// TwinCAT 3 PLC project kfe_rix_motion
// Title: plc-kfe-rix-motion
// Company: SLAC
// ProjectVersion: 0.0.0
// ProgramVersion: 3.1.4022.7
// CompilerDefines: K
// libraries:
//   LCLS General, * (SLAC)
//   lcls-twincat-common-components, * (SLAC)
//   lcls-twincat-motion, * (SLAC)
//   lcls-twincat-physics, * (SLAC)
//   PMPS, * (SLAC - LCLS)
//   Tc2_Standard, * (Beckhoff Automation GmbH)
//   Tc2_System, * (Beckhoff Automation GmbH)
//   Tc3_Module, * (Beckhoff Automation GmbH)
// project tree:
//   DUTs/ DUT_SATT_Filter.TcDUT (not stored), ENUM_SXR_SATT_Position.TcDUT (not stored)
//   GVLs/ GVL.TcGVL (not stored), Main.TcGVL (not stored)
//   / PlcTask.TcTTO (not stored)
//   POUs/AT1K2/ FB_AT1K2.TcPOU (not stored)
//   POUs/AT2K2/ FB_AttenuatorElementDensity.TcPOU (not stored), FB_SXR_SATT_PositionState.TcPOU (not stored), FB_SXR_SATT_Stage.TcPOU (not stored)
//   POUs/ PRG_1_PlcTask.TcPOU (not stored), PRG_2_PMPS_PRE.TcPOU (not stored), PRG_3_PMPS_POST.TcPOU (not stored), PRG_4_LOG.TcPOU (not stored), PRG_AT1K2_SOLID.TcPOU (not stored), PRG_AT2K2_SOLID.TcPOU (not stored), PRG_IM6K2_PPM.TcPOU, PRG_LI3K2_K2B.TcPOU, PRG_PF1K2_WFS.TcPOU, PRG_LI2K2_K2A.TcPOU, PRG_IM1K1_PPM.TcPOU, PRG_AL1K2_L2SI.TcPOU, PRG_IM2K2_PPM.TcPOU, PRG_IM2K1_PPM.TcPOU, PRG_IM1K2_PPM.TcPOU, PRG_IM3K2_PPM.TcPOU, PRG_IM4K2_PPM.TcPOU, PRG_IM5K2_PPM.TcPOU, PRG_PF2K2_WFS.TcPOU, PRG_TM1K2_ATM.TcPOU, PRG_TM2K2_ATM.TcPOU (not stored), PRG_ST3K2_TERM.TcPOU (not stored)
//   POUs/TM2K2/ ENUM_TM2K2_States.TcDUT (not stored), FB_TM2K2.TcPOU (not stored), FB_TM2K2_States.TcPOU (not stored)

// ---- POUs/PRG_IM6K2_PPM.TcPOU
PROGRAM PRG_IM6K2_PPM
VAR
    {attribute 'pytmc' := '
        pv: IM6K2:PPM
        io: io
    '}
    {attribute 'TcLinkTo' := '.fbGige.iIlluminatorINT := TIIB[IM6K2-EL4004-E7]^AO Outputs Channel 1^Analog output;
                              .fbGige.bGigePower := TIIB[IM6K2-EL2004-E3]^Channel 2^Output;
                              .fbPowerMeter.iVoltageINT := TIIB[IM6K2-EL3062-E6]^AI Standard Channel 1^Value;
                              .fbPowerMeter.fbThermoCouple.bError := TIIB[IM6K2-EL3314-E4]^TC Inputs Channel 1^Status^Error;
                              .fbPowerMeter.fbThermoCouple.bUnderrange := TIIB[IM6K2-EL3314-E4]^TC Inputs Channel 1^Status^Underrange;
                              .fbPowerMeter.fbThermoCouple.bOverrange := TIIB[IM6K2-EL3314-E4]^TC Inputs Channel 1^Status^Overrange;
                              .fbPowerMeter.fbThermoCouple.iRaw := TIIB[IM6K2-EL3314-E4]^TC Inputs Channel 1^Value;
                              .fbYagThermoCouple.bError := TIIB[IM6K2-EL3314-E4]^TC Inputs Channel 2^Status^Error;
                              .fbYagThermoCouple.bUnderrange := TIIB[IM6K2-EL3314-E4]^TC Inputs Channel 2^Status^Underrange;
                              .fbYagThermoCouple.bOverrange := TIIB[IM6K2-EL3314-E4]^TC Inputs Channel 2^Status^Overrange;
                              .fbYagThermoCouple.iRaw 6K2-EL3314-E4]^TC Inputs Channel 2^Value;
                              .fbFlowMeter.iRaw := TIIB[IM1K2-EL3052-E5]^AI Standard Channel 1^Value'}
    fbIM6K2: FB_PPM;
END_VAR


fbIM6K2.stOut.fPosition := -8.61;
fbIM6K2.stOut.bUseRawCounts := FALSE;
fbIM6K2.stOut.bValid := TRUE;
fbIM6K2.stOut.stPMPS.sPmpsState := 'IM6K2:PPM-OUT';

fbIM6K2.stPower.fPosition := -47.71;
fbIM6K2.stPower.bUseRawCounts := FALSE;
fbIM6K2.stPower.bValid := TRUE;
fbIM6K2.stPower.stPMPS.sPmpsState := 'IM6K2:PPM-POWERMETER';

fbIM6K2.stYag1.fPosition := -71.71;
fbIM6K2.stYag1.bUseRawCounts := FALSE;
fbIM6K2.stYag1.bValid := TRUE;
fbIM6K2.stYag1.stPMPS.sPmpsState := 'IM6K2:PPM-YAG1';

fbIM6K2.stYag2.fPosition := -97.72;
fbIM6K2.stYag2.bUseRawCounts := FALSE;
fbIM6K2.stYag2.bValid := TRUE;
fbIM6K2.stYag2.stPMPS.sPmpsState := 'IM6K2:PPM-YAG2';

fbIM6K2(
    fbArbiter := GVL.fbArbiter2,
    fbFFHWO := GVL.fbFastFaultOutput2,
    stYStage := Main.M24,
    sDeviceName := 'IM6K2:PPM',
    sTransitionKey := 'IM6K2:PPM-TRANSITION',
    bEnableMotion := TRUE,
    bEnableBeamParams := TRUE,
    bEnablePositionLimits := TRUE,
    fFlowOffset := 0.0,
);

END_PROGRAM

// ---- POUs/PRG_LI3K2_K2B.TcPOU
PROGRAM PRG_LI3K2_K2B
VAR
    {attribute 'pytmc' := '
        pv: LI3K2:K2B
        io: io
    '}
    fbLI3K2: FB_LIC;

    //stSiBP: ST_BeamParams := PMPS_GVL.cstFullBeam;
    //stFoilBP: ST_BeamParams := PMPS_GVL.cstFullBeam;
END_VAR

(*
   Avoid damage peak between 3.2 keV and 1.6 keV
*)
//stSiBp.neVRange := F_eVExcludeRange(1600, 3200);
// Drop transmission to 20%
//stSiBP.nTran := 0.2;

// Drop transmission to 10%
//stFoilBP.nTran := 0.1;

fbLI3K2.stOut.fPosition := 0.118;
fbLI3K2.stOut.bUseRawCounts := FALSE;
fbLI3K2.stOut.bValid := TRUE;
fbLI3K2.stOut.stPMPS.sPmpsState := 'LI3K2:K2B-OUT';

fbLI3K2.stMirror1.fPosition := -36.38;
fbLI3K2.stMirror1.bUseRawCounts := FALSE;
fbLI3K2.stMirror1.bValid := TRUE;
fbLI3K2.stMirror1.stPMPS.sPmpsState := 'LI3K2:K2B-MIRROR1';

fbLI3K2.stMirror2.fPosition := -70.38;
fbLI3K2.stMirror2.bUseRawCounts := FALSE;
fbLI3K2.stMirror2.bValid := TRUE;
fbLI3K2.stMirror2.stPMPS.sPmpsState := 'LI3K2:K2B-MIRROR2';

fbLI3K2.stTarget1.fPosition := -102.38;
fbLI3K2.stTarget1.bUseRawCounts := FALSE;
fbLI3K2.stTarget1.bValid := TRUE;
fbLI3K2.stTarget1.stPMPS.sPmpsState := 'LI3K2:K2B-TARGET1';

fbLI3K2(
    fbArbiter := GVL.fbArbiter2,
    fbFFHWO := GVL.fbFastFaultOutput2,
    stYStage := Main.M21,
    sDeviceName := 'LI3K2:K2B',
    sTransitionKey := 'LI3K2:K2B-TRANSITION',
    bEnableMotion := TRUE,
    bEnableBeamParams := TRUE,
    bEnablePositionLimits := TRUE,
);

END_PROGRAM

// ---- POUs/PRG_PF1K2_WFS.TcPOU
PROGRAM PRG_PF1K2_WFS
VAR
    {attribute 'pytmc' := '
        pv: PF1K2:WFS
        io: io
    '}
    {attribute 'TcLinkTo' := '.fbThermoCouple1.bError 		:= TIIB[PF1K2-EL3314-E5]^TC Inputs Channel 1^Status^Error;
                              .fbThermoCouple1.bUnderrange	:= TIIB[PF1K2-EL3314-E5]^TC Inputs Channel 1^Status^Underrange;
                              .fbThermoCouple1.bOverrange 	:= TIIB[PF1K2-EL3314-E5]^TC Inputs Channel 1^Status^Overrange;
                              .fbThermoCouple1.iRaw 		:= TIIB[PF1K2-EL3314-E5]^TC Inputs Channel 1^Value;
                              .fbThermoCouple2.bError 		:= TIIB[PF1K2-EL3314-E5]^TC Inputs Channel 2^Status^Error;
                              .fbThermoCouple2.bUnderrange 	:= TIIB[PF1K2-EL3314-E5]^TC Inputs Channel 2^Status^Underrange;
                              .fbThermoCouple2.bOverrange 	:= TIIB[PF1K2-EL3314-E5]^TC Inputs Channel 2^Status^Overrange;
                              .fbThermoCouple2.iRaw 		:= TIIB[PF1K2-EL3314-E5]^TC Inputs Channel 2^Value'}
    fbPF1K2: FB_WFS;

    //stSiBP: ST_BeamParams := PMPS_GVL.cstFullBeam;
END_VAR

(*
   Avoid damage peak between 3.2 keV and 1.6 keV
*)
//stSiBp.neVRange := F_eVExcludeRange(1600, 3200);
// Drop transmission to 20%
//stSiBP.nTran := 0.2;

fbPF1K2.stOut.fPosition := -13.00;
fbPF1K2.stOut.bUseRawCounts := FALSE;
fbPF1K2.stOut.bValid := TRUE;
fbPF1K2.stOut.stPMPS.sPmpsState := 'PF1K2:WFS-OUT';

fbPF1K2.stTarget1.fPosition := -97.13;
fbPF1K2.stTarget1.bUseRawCounts := FALSE;
fbPF1K2.stTarget1.bValid := TRUE;
fbPF1K2.stTarget1.stPMPS.sPmpsState := 'PF1K2:WFS-TARGET1';

fbPF1K2.stTarget2.fPosition := -82.755;
fbPF1K2.stTarget2.bUseRawCounts := FALSE;
fbPF1K2.stTarget2.bValid := TRUE;
fbPF1K2.stTarget2.stPMPS.sPmpsState := 'PF1K2:WFS-TARGET2';

fbPF1K2.stTarget3.fPosition := -68.38;
fbPF1K2.stTarget3.bUseRawCounts := FALSE;
fbPF1K2.stTarget3.bValid := TRUE;
fbPF1K2.stTarget3.stPMPS.sPmpsState := 'PF1K2:WFS-TARGET3';

fbPF1K2.stTarget4.fPosition := -54.004;
fbPF1K2.stTarget4.bUseRawCounts := FALSE;
fbPF1K2.stTarget4.bValid := TRUE;
fbPF1K2.stTarget4.stPMPS.sPmpsState := 'PF1K2:WFS-TARGET4';

fbPF1K2.stTarget5.fPosition := -39.629;
fbPF1K2.stTarget5.bUseRawCounts := FALSE;
fbPF1K2.stTarget5.bValid := TRUE;
fbPF1K2.stTarget5.stPMPS.sPmpsState := 'PF1K2:WFS-TARGET5';

fbPF1K2(
    fbArbiter := GVL.fbArbiter2,
    fbFFHWO := GVL.fbFastFaultOutput2,
    stYStage := Main.M12,
    stZStage := Main.M13,
    sDeviceName := 'PF1K2:WFS',
    sTransitionKey := 'PF1K2:WFS-TRANSITION',
    bEnableMotion := TRUE,
    bEnableBeamParams := TRUE,
    bEnablePositionLimits := TRUE,
);

END_PROGRAM

// ---- POUs/PRG_LI2K2_K2A.TcPOU
PROGRAM PRG_LI2K2_K2A
VAR
    {attribute 'pytmc' := '
        pv: LI2K2:K2A
        io: io
    '}
    fbLI2K2: FB_LIC;

    //stSiBP: ST_BeamParams := PMPS_GVL.cstFullBeam;
    //stFoilBP: ST_BeamParams := PMPS_GVL.cstFullBeam;
END_VAR

(*
   Avoid damage peak between 3.2 keV and 1.6 keV
*)
//stSiBp.neVRange := F_eVExcludeRange(1600, 3200);
// Drop transmission to 20%
//stSiBP.nTran := 0.2;

// Drop transmission to 10%
////stFoilBP.nTran := 0.1;

fbLI2K2.stOut.fPosition := 1.2;
fbLI2K2.stOut.bUseRawCounts := FALSE;
fbLI2K2.stOut.bValid := TRUE;
fbLI2K2.stOut.stPMPS.sPmpsState := 'LI2K2:K2A-OUT';

fbLI2K2.stMirror1.fPosition := -35.3;
fbLI2K2.stMirror1.bUseRawCounts := FALSE;
fbLI2K2.stMirror1.bValid := TRUE;
fbLI2K2.stMirror1.stPMPS.sPmpsState := 'LI2K2:K2A-MIRROR1';

fbLI2K2.stMirror2.fPosition := -69.3;
fbLI2K2.stMirror2.bUseRawCounts := FALSE;
fbLI2K2.stMirror2.bValid := TRUE;
fbLI2K2.stMirror2.stPMPS.sPmpsState := 'LI2K2:K2A-MIRROR2';

fbLI2K2.stTarget1.fPosition := -101.3;
fbLI2K2.stTarget1.bUseRawCounts := FALSE;
fbLI2K2.stTarget1.bValid := TRUE;
fbLI2K2.stTarget1.stPMPS.sPmpsState := 'LI2K2:K2A-TARGET1';

fbLI2K2(
    fbArbiter := GVL.fbArbiter2,
    fbFFHWO := GVL.fbFastFaultOutput2,
    stYStage := Main.M11,
    sDeviceName := 'LI2K2:K2A',
    sTransitionKey := 'LI2K2:K2A-TRANSITION',
    bEnableMotion := TRUE,
    bEnableBeamParams := TRUE,
    bEnablePositionLimits := TRUE,
);

END_PROGRAM

// ---- POUs/PRG_IM1K1_PPM.TcPOU
PROGRAM PRG_IM1K1_PPM
VAR
    {attribute 'pytmc' := '
        pv: IM1K1:PPM
        io: io
    '}
    {attribute 'TcLinkTo' := '.fbGige.iIlluminatorINT := TIIB[IM1K1-EL4004]^AO Outputs Channel 1^Analog output;
                              .fbGige.bGigePower := TIIB[IM1K1-EL2004]^Channel 2^Output;
                              .fbPowerMeter.iVoltageINT := TIIB[IM1K1-EL3062]^AI Standard Channel 1^Value;
                              .fbPowerMeter.fbThermoCouple.bError := TIIB[IM1K1-EL3314]^TC Inputs Channel 1^Status^Error;
                              .fbPowerMeter.fbThermoCouple.bUnderrange := TIIB[IM1K1-EL3314]^TC Inputs Channel 1^Status^Underrange;
                              .fbPowerMeter.fbThermoCouple.bOverrange := TIIB[IM1K1-EL3314]^TC Inputs Channel 1^Status^Overrange;
                              .fbPowerMeter.fbThermoCouple.iRaw := TIIB[IM1K1-EL3314]^TC Inputs Channel 1^Value;
                              .fbYagThermoCouple.bError := TIIB[IM1K1-EL3314]^TC Inputs Channel 2^Status^Error;
                              .fbYagThermoCouple.bUnderrange := TIIB[IM1K1-EL3314]^TC Inputs Channel 2^Status^Underrange;
                              .fbYagThermoCouple.bOverrange := TIIB[IM1K1-EL3314]^TC Inputs Channel 2^Status^Overrange;
                              .fbYagThermoCouple.iRaw := TIIB[IM1K1-EL3314]^TC Inputs Channel 2^Value'}
    fbIM1K1: FB_PPM;
END_VAR

fbIM1K1.stOut.fPosition := -8.82;
fbIM1K1.stOut.bUseRawCounts := FALSE;
fbIM1K1.stOut.bValid := TRUE;
fbIM1K1.stOut.stPMPS.sPmpsState := 'IM1K1:PPM-OUT';

fbIM1K1.stPower.fPosition := -47.92;
fbIM1K1.stPower.bUseRawCounts := FALSE;
fbIM1K1.stPower.bValid := TRUE;
fbIM1K1.stPower.stPMPS.sPmpsState := 'IM1K1:PPM-POWERMETER';

fbIM1K1.stYag1.fPosition := -71.92;
fbIM1K1.stYag1.bUseRawCounts := FALSE;
fbIM1K1.stYag1.bValid := TRUE;
fbIM1K1.stYag1.stPMPS.sPmpsState := 'IM1K1:PPM-YAG1';

fbIM1K1.stYag2.fPosition := -97.93;
fbIM1K1.stYag2.bUseRawCounts := FALSE;
fbIM1K1.stYag2.bValid := TRUE;
fbIM1K1.stYag2.stPMPS.sPmpsState := 'IM1K1:PPM-YAG2';

fbIM1K1(
    fbArbiter := GVL.fbArbiter1,
    fbFFHWO := GVL.fbFastFaultOutput1,
    stYStage := Main.M1,
    sDeviceName := 'IM1K1:PPM',
    sTransitionKey := 'IM1K1:PPM-TRANSITION',
    bEnableMotion := TRUE,
    bEnableBeamParams := TRUE,
    bEnablePositionLimits := FALSE,
    fFlowOffset := 0.0,
);

END_PROGRAM

// ---- POUs/PRG_AL1K2_L2SI.TcPOU
PROGRAM PRG_AL1K2_L2SI
VAR
    {attribute 'pytmc' := '
        pv: AL1K2:L2SI
        io: io
    '}
    {attribute 'TcLinkTo' := '.fbLaser.iLaserINT := TIIB[AL1K2-EL4004-E4]^AO Outputs Channel 1^Analog output;
                              .fbLaser.iShutdownINT := TIIB[AL1K2-EL4004-E4]^AO Outputs Channel 2^Analog output'}
    fbAL1K2: FB_REF;
END_VAR


fbAL1K2.stOut.fPosition := -33.5; // Upper limit
fbAL1K2.stOut.bUseRawCounts := FALSE;
fbAL1K2.stOut.bValid := TRUE;
fbAL1K2.stOut.stPMPS.sPmpsState := 'AL1K2:L2SI-OUT';

fbAL1K2.stIn.fPosition := -75; // Current position at time of edit
fbAL1K2.stIn.bUseRawCounts := FALSE;
fbAL1K2.stIn.bValid := TRUE;
fbAL1K2.stIn.stPMPS.sPmpsState := 'AL1K2:L2SI-IN';

fbAL1K2(
    stYStage := Main.M5,
    fbArbiter := GVL.fbArbiter2,
    fbFFHWO := GVL.fbFastFaultOutput2,
    sDeviceName := 'AL1K2:L2SI',
    sTransitionKey := 'AL1K2:L2SI-TRANSITION',
    bEnableMotion := TRUE,
    bEnableBeamParams := TRUE,
    bEnablePositionLimits := TRUE
);

END_PROGRAM

// ---- POUs/PRG_IM2K2_PPM.TcPOU
PROGRAM PRG_IM2K2_PPM
VAR
    {attribute 'pytmc' := '
        pv: IM2K2:PPM
        io: io
    '}
    {attribute 'TcLinkTo' := '.fbGige.iIlluminatorINT := TIIB[IM2K2-EL4004-E7]^AO Outputs Channel 1^Analog output;
                              .fbGige.bGigePower := TIIB[IM2K2-EL2004-E3]^Channel 2^Output;
                              .fbPowerMeter.iVoltageINT := TIIB[IM2K2-EL3062-E6]^AI Standard Channel 1^Value;
                              .fbPowerMeter.fbThermoCouple.bError := TIIB[IM2K2-EL3314-E4]^TC Inputs Channel 1^Status^Error;
                              .fbPowerMeter.fbThermoCouple.bUnderrange := TIIB[IM2K2-EL3314-E4]^TC Inputs Channel 1^Status^Underrange;
                              .fbPowerMeter.fbThermoCouple.bOverrange := TIIB[IM2K2-EL3314-E4]^TC Inputs Channel 1^Status^Overrange;
                              .fbPowerMeter.fbThermoCouple.iRaw := TIIB[IM2K2-EL3314-E4]^TC Inputs Channel 1^Value;
                              .fbYagThermoCouple.bError := TIIB[IM2K2-EL3314-E4]^TC Inputs Channel 2^Status^Error;
                              .fbYagThermoCouple.bUnderrange := TIIB[IM2K2-EL3314-E4]^TC Inputs Channel 2^Status^Underrange;
                              .fbYagThermoCouple.bOverrange := TIIB[IM2K2-EL3314-E4]^TC Inputs Channel 2^Status^Overrange;
                              .fbYagThermoCouple.iRaw := TIIB[IM2K2-EL3314-E4]^TC Inputs Channel 2^Value;
                              .fbFlowMeter.iRaw := TIIB[IM1K2-EL3052-E5]^AI Standard Channel 1^Value'}  //IM1/2/3/4K2 same flow meter
    fbIM2K2: FB_PPM;
END_VAR


fbIM2K2.stOut.fPosition := -8.49;
fbIM2K2.stOut.bUseRawCounts := FALSE;
fbIM2K2.stOut.bValid := TRUE;
fbIM2K2.stOut.stPMPS.sPmpsState := 'IM2K2:PPM-OUT';

fbIM2K2.stPower.fPosition := -47.59;
fbIM2K2.stPower.bUseRawCounts := FALSE;
fbIM2K2.stPower.bValid := TRUE;
fbIM2K2.stPower.stPMPS.sPmpsState := 'IM2K2:PPM-POWERMETER';

fbIM2K2.stYag1.fPosition := -71.59;
fbIM2K2.stYag1.bUseRawCounts := FALSE;
fbIM2K2.stYag1.bValid := TRUE;
fbIM2K2.stYag1.stPMPS.sPmpsState := 'IM2K2:PPM-YAG1';

fbIM2K2.stYag2.fPosition := -97.60;
fbIM2K2.stYag2.bUseRawCounts := FALSE;
fbIM2K2.stYag2.bValid := TRUE;
fbIM2K2.stYag2.stPMPS.sPmpsState := 'IM2K2:PPM-YAG2';

fbIM2K2(
    fbArbiter := GVL.fbArbiter2,
    fbFFHWO := GVL.fbFastFaultOutput2,
    stYStage := Main.M6,
    sDeviceName := 'IM2K2:PPM',
    sTransitionKey := 'IM2K2:PPM-TRANSITION',
    bEnableMotion := TRUE,
    bEnableBeamParams := TRUE,
    bEnablePositionLimits := TRUE,
);

END_PROGRAM

// ---- POUs/PRG_IM2K1_PPM.TcPOU
PROGRAM PRG_IM2K1_PPM
VAR
    {attribute 'pytmc' := '
        pv: IM2K1:PPM
        io: io
    '}
    {attribute 'TcLinkTo' := '.fbGige.iIlluminatorINT := TIIB[IM2K1-EL4004]^AO Outputs Channel 1^Analog output;
                              .fbGige.bGigePower := TIIB[IM2K1-EL2004]^Channel 2^Output;
                              .fbPowerMeter.iVoltageINT := TIIB[IM2K1-EL3062]^AI Standard Channel 1^Value;
                              .fbPowerMeter.fbThermoCouple.bError := TIIB[IM2K1-EL3314]^TC Inputs Channel 1^Status^Error;
                              .fbPowerMeter.fbThermoCouple.bUnderrange := TIIB[IM2K1-EL3314]^TC Inputs Channel 1^Status^Underrange;
                              .fbPowerMeter.fbThermoCouple.bOverrange := TIIB[IM2K1-EL3314]^TC Inputs Channel 1^Status^Overrange;
                              .fbPowerMeter.fbThermoCouple.iRaw := TIIB[IM2K1-EL3314]^TC Inputs Channel 1^Value;
                              .fbYagThermoCouple.bError := TIIB[IM2K1-EL3314]^TC Inputs Channel 2^Status^Error;
                              .fbYagThermoCouple.bUnderrange := TIIB[IM2K1-EL3314]^TC Inputs Channel 2^Status^Underrange;
                              .fbYagThermoCouple.bOverrange := TIIB[IM2K1-EL3314]^TC Inputs Channel 2^Status^Overrange;
                              .fbYagThermoCouple.iRaw := TIIB[IM2K1-EL3314]^TC Inputs Channel 2^Value'}
    fbIM2K1: FB_PPM;
END_VAR


fbIM2K1.stOut.fPosition := -9.09;
fbIM2K1.stOut.bUseRawCounts := FALSE;
fbIM2K1.stOut.bValid := TRUE;
fbIM2K1.stOut.stPMPS.sPmpsState := 'IM2K1:PPM-OUT';

fbIM2K1.stPower.fPosition := -48.19;
fbIM2K1.stPower.bUseRawCounts := FALSE;
fbIM2K1.stPower.bValid := TRUE;
fbIM2K1.stPower.stPMPS.sPmpsState := 'IM2K1:PPM-POWERMETER';

fbIM2K1.stYag1.fPosition := -72.19;
fbIM2K1.stYag1.bUseRawCounts := FALSE;
fbIM2K1.stYag1.bValid := TRUE;
fbIM2K1.stYag1.stPMPS.sPmpsState := 'IM2K1:PPM-YAG1';

fbIM2K1.stYag2.fPosition := -98.2;
fbIM2K1.stYag2.bUseRawCounts := FALSE;
fbIM2K1.stYag2.bValid := TRUE;
fbIM2K1.stYag2.stPMPS.sPmpsState := 'IM2K1:PPM-YAG2';

fbIM2K1(
    fbArbiter := GVL.fbArbiter1,
    fbFFHWO := GVL.fbFastFaultOutput1,
    stYStage := Main.M2,
    sDeviceName := 'IM2K1:PPM',
    sTransitionKey := 'IM2K1:PPM-TRANSITION',
    bEnableMotion := TRUE,
    bEnableBeamParams := TRUE,
    bEnablePositionLimits := TRUE,
    fFlowOffset := 0.0,
);

END_PROGRAM

// ---- POUs/PRG_IM1K2_PPM.TcPOU
PROGRAM PRG_IM1K2_PPM
VAR
    {attribute 'pytmc' := '
        pv: IM1K2:PPM
        io: io
    '}
    {attribute 'TcLinkTo' := '.fbGige.iIlluminatorINT := TIIB[IM1K2-EL4004-E7]^AO Outputs Channel 1^Analog output;
                              .fbGige.bGigePower := TIIB[IM1K2-EL2004-E3]^Channel 2^Output;
                              .fbPowerMeter.iVoltageINT := TIIB[IM1K2-EL3062-E6]^AI Standard Channel 1^Value;
                              .fbPowerMeter.fbThermoCouple.bError := TIIB[IM1K2-EL3314-E4]^TC Inputs Channel 1^Status^Error;
                              .fbPowerMeter.fbThermoCouple.bUnderrange := TIIB[IM1K2-EL3314-E4]^TC Inputs Channel 1^Status^Underrange;
                              .fbPowerMeter.fbThermoCouple.bOverrange := TIIB[IM1K2-EL3314-E4]^TC Inputs Channel 1^Status^Overrange;
                              .fbPowerMeter.fbThermoCouple.iRaw := TIIB[IM1K2-EL3314-E4]^TC Inputs Channel 1^Value;
                              .fbYagThermoCouple.bError := TIIB[IM1K2-EL3314-E4]^TC Inputs Channel 2^Status^Error;
                              .fbYagThermoCouple.bUnderrange := TIIB[IM1K2-EL3314-E4]^TC Inputs Channel 2^Status^Underrange;
                              .fbYagThermoCouple.bOverrange := TIIB[IM1K2-EL3314-E4]^TC Inputs Channel 2^Status^Overrange;
                              .fbYagThermoCouple.iRaw := TIIB[IM1K2-EL3314-E4]^TC Inputs Channel 2^Value;
                              .fbFlowMeter.iRaw := TIIB[IM1K2-EL3052-E5]^AI Standard Channel 1^Value'}
    fbIM1K2: FB_PPM;
END_VAR

fbIM1K2.stOut.fPosition := -9.82;
fbIM1K2.stOut.bUseRawCounts := FALSE;
fbIM1K2.stOut.bValid := TRUE;
fbIM1K2.stOut.stPMPS.sPmpsState := 'IM1K2:PPM-OUT';

fbIM1K2.stPower.fPosition := -48.92;
fbIM1K2.stPower.bUseRawCounts := FALSE;
fbIM1K2.stPower.bValid := TRUE;
fbIM1K2.stPower.stPMPS.sPmpsState := 'IM1K2:PPM-POWERMETER';

fbIM1K2.stYag1.fPosition := -72.92;
fbIM1K2.stYag1.bUseRawCounts := FALSE;
fbIM1K2.stYag1.bValid := TRUE;
fbIM1K2.stYag1.stPMPS.sPmpsState := 'IM1K2:PPM-YAG1';

fbIM1K2.stYag2.fPosition := -98.93;
fbIM1K2.stYag2.bUseRawCounts := FALSE;
fbIM1K2.stYag2.bValid := TRUE;
fbIM1K2.stYag2.stPMPS.sPmpsState := 'IM1K2:PPM-YAG2';

fbIM1K2(
    fbArbiter := GVL.fbArbiter1,
    fbFFHWO := GVL.fbFastFaultOutput1,
    stYStage := Main.M4,
    sDeviceName := 'IM1K2:PPM',
    sTransitionKey := 'IM1K2:PPM-TRANSITION',
    bEnableMotion := TRUE,
    bEnableBeamParams := TRUE,
    bEnablePositionLimits := TRUE,
);

END_PROGRAM

// ---- POUs/PRG_IM3K2_PPM.TcPOU
PROGRAM PRG_IM3K2_PPM
VAR
    {attribute 'pytmc' := '
        pv: IM3K2:PPM
        io: io
    '}
    {attribute 'TcLinkTo' := '.fbGige.iIlluminatorINT := TIIB[IM3K2-EL4004-E7]^AO Outputs Channel 1^Analog output;
                              .fbGige.bGigePower := TIIB[IM3K2-EL2004-E3]^Channel 2^Output;
                              .fbPowerMeter.iVoltageINT := TIIB[IM3K2-EL3062-E6]^AI Standard Channel 1^Value;
                              .fbPowerMeter.fbThermoCouple.bError := TIIB[IM3K2-EL3314-E4]^TC Inputs Channel 1^Status^Error;
                              .fbPowerMeter.fbThermoCouple.bUnderrange := TIIB[IM3K2-EL3314-E4]^TC Inputs Channel 1^Status^Underrange;
                              .fbPowerMeter.fbThermoCouple.bOverrange := TIIB[IM3K2-EL3314-E4]^TC Inputs Channel 1^Status^Overrange;
                              .fbPowerMeter.fbThermoCouple.iRaw := TIIB[IM3K2-EL3314-E4]^TC Inputs Channel 1^Value;
                              .fbYagThermoCouple.bError := TIIB[IM3K2-EL3314-E4]^TC Inputs Channel 2^Status^Error;
                              .fbYagThermoCouple.bUnderrange := TIIB[IM3K2-EL3314-E4]^TC Inputs Channel 2^Status^Underrange;
                              .fbYagThermoCouple.bOverrange := TIIB[IM3K2-EL3314-E4]^TC Inputs Channel 2^Status^Overrange;
                              .fbYagThermoCouple.iRaw := TIIB[IM3K2-EL3314-E4]^TC Inputs Channel 2^Value;
                              .fbFlowMeter.iRaw := TIIB[IM1K2-EL3052-E5]^AI Standard Channel 1^Value'}  //IM1/2/3/4K2 same flow meter
    fbIM3K2: FB_PPM;
END_VAR


fbIM3K2.stOut.fPosition := -9.61;
fbIM3K2.stOut.bUseRawCounts := FALSE;
fbIM3K2.stOut.bValid := TRUE;
fbIM3K2.stOut.stPMPS.sPmpsState := 'IM3K2:PPM-OUT';

fbIM3K2.stPower.fPosition := -48.71;
fbIM3K2.stPower.bUseRawCounts := FALSE;
fbIM3K2.stPower.bValid := TRUE;
fbIM3K2.stPower.stPMPS.sPmpsState := 'IM3K2:PPM-POWERMETER';

fbIM3K2.stYag1.fPosition := -72.71;
fbIM3K2.stYag1.bUseRawCounts := FALSE;
fbIM3K2.stYag1.bValid := TRUE;
fbIM3K2.stYag1.stPMPS.sPmpsState := 'IM3K2:PPM-YAG1';

fbIM3K2.stYag2.fPosition := -98.72;
fbIM3K2.stYag2.bUseRawCounts := FALSE;
fbIM3K2.stYag2.bValid := TRUE;
fbIM3K2.stYag2.stPMPS.sPmpsState := 'IM3K2:PPM-YAG2';

fbIM3K2(
    fbArbiter := GVL.fbArbiter2,
    fbFFHWO := GVL.fbFastFaultOutput2,
    stYStage := Main.M7,
    sDeviceName := 'IM3K2:PPM',
    sTransitionKey := 'IM3K2:PPM-TRANSITION',
    bEnableMotion := TRUE,
    bEnableBeamParams := TRUE,
    bEnablePositionLimits := TRUE,
    fFlowOffset := 0.0,
);

END_PROGRAM

// ---- POUs/PRG_IM4K2_PPM.TcPOU
PROGRAM PRG_IM4K2_PPM
VAR
    {attribute 'pytmc' := '
        pv: IM4K2:PPM
        io: io
    '}
     {attribute 'TcLinkTo' := '.fbGige.iIlluminatorINT := TIIB[IM4K2-EL4004-E7]^AO Outputs Channel 1^Analog output;
                              .fbGige.bGigePower := TIIB[IM4K2-EL2004-E3]^Channel 2^Output;
                              .fbPowerMeter.iVoltageINT := TIIB[IM4K2-EL3062-E6]^AI Standard Channel 1^Value;
                              .fbPowerMeter.fbThermoCouple.bError := TIIB[IM4K2-EL3314-E4]^TC Inputs Channel 1^Status^Error;
                              .fbPowerMeter.fbThermoCouple.bUnderrange := TIIB[IM4K2-EL3314-E4]^TC Inputs Channel 1^Status^Underrange;
                              .fbPowerMeter.fbThermoCouple.bOverrange := TIIB[IM4K2-EL3314-E4]^TC Inputs Channel 1^Status^Overrange;
                              .fbPowerMeter.fbThermoCouple.iRaw := TIIB[IM4K2-EL3314-E4]^TC Inputs Channel 1^Value;
                              .fbYagThermoCouple.bError := TIIB[IM4K2-EL3314-E4]^TC Inputs Channel 2^Status^Error;
                              .fbYagThermoCouple.bUnderrange := TIIB[IM4K2-EL3314-E4]^TC Inputs Channel 2^Status^Underrange;
                              .fbYagThermoCouple.bOverrange := TIIB[IM4K2-EL3314-E4]^TC Inputs Channel 2^Status^Overrange;
                              .fbYagThermoCouple.iRaw := TIIB[IM4K2-EL3314-E4]^TC Inputs Channel 2^Value;
                              .fbFlowMeter.iRaw := TIIB[IM1K2-EL3052-E5]^AI Standard Channel 1^Value'}  //IM1/2/3/4K2 same flow meter
    fbIM4K2: FB_PPM;
END_VAR


fbIM4K2.stOut.fPosition := -10.80;
fbIM4K2.stOut.bUseRawCounts := FALSE;
fbIM4K2.stOut.bValid := TRUE;
fbIM4K2.stOut.stPMPS.sPmpsState := 'IM4K2:PPM-OUT';

fbIM4K2.stPower.fPosition := -49.90;
fbIM4K2.stPower.bUseRawCounts := FALSE;
fbIM4K2.stPower.bValid := TRUE;
fbIM4K2.stPower.stPMPS.sPmpsState := 'IM4K2:PPM-POWERMETER';

fbIM4K2.stYag1.fPosition := -73.90;
fbIM4K2.stYag1.bUseRawCounts := FALSE;
fbIM4K2.stYag1.bValid := TRUE;
fbIM4K2.stYag1.stPMPS.sPmpsState := 'IM4K2:PPM-YAG1';

fbIM4K2.stYag2.fPosition := -99.91;
fbIM4K2.stYag2.bUseRawCounts := FALSE;
fbIM4K2.stYag2.bValid := TRUE;
fbIM4K2.stYag2.stPMPS.sPmpsState := 'IM4K2:PPM-YAG2';

fbIM4K2(
    fbArbiter := GVL.fbArbiter2,
    fbFFHWO := GVL.fbFastFaultOutput2,
    stYStage := Main.M8,
    sDeviceName := 'IM4K2:PPM',
    sTransitionKey := 'IM4K2:PPM-TRANSITION',
    bEnableMotion := TRUE,
    bEnableBeamParams := TRUE,
    bEnablePositionLimits := TRUE,
    fFlowOffset := 0.0,
);

END_PROGRAM

// ---- POUs/PRG_IM5K2_PPM.TcPOU
PROGRAM PRG_IM5K2_PPM
VAR
    {attribute 'pytmc' := '
        pv: IM5K2:PPM
        io: io
    '}
    {attribute 'TcLinkTo' := '.fbGige.iIlluminatorINT := TIIB[IM5K2-EL4004-E7]^AO Outputs Channel 1^Analog output;
                              .fbGige.bGigePower := TIIB[IM5K2-EL2004-E3]^Channel 2^Output;
                              .fbPowerMeter.iVoltageINT := TIIB[IM5K2-EL3062-E6]^AI Standard Channel 1^Value;
                              .fbPowerMeter.fbThermoCouple.bError := TIIB[IM5K2-EL3314-E4]^TC Inputs Channel 1^Status^Error;
                              .fbPowerMeter.fbThermoCouple.bUnderrange := TIIB[IM5K2-EL3314-E4]^TC Inputs Channel 1^Status^Underrange;
                              .fbPowerMeter.fbThermoCouple.bOverrange := TIIB[IM5K2-EL3314-E4]^TC Inputs Channel 1^Status^Overrange;
                              .fbPowerMeter.fbThermoCouple.iRaw := TIIB[IM5K2-EL3314-E4]^TC Inputs Channel 1^Value;
                              .fbYagThermoCouple.bError := TIIB[IM5K2-EL3314-E4]^TC Inputs Channel 2^Status^Error;
                              .fbYagThermoCouple.bUnderrange := TIIB[IM5K2-EL3314-E4]^TC Inputs Channel 2^Status^Underrange;
                              .fbYagThermoCouple.bOverrange := TIIB[IM5K2-EL3314-E4]^TC Inputs Channel 2^Status^Overrange;
                              .fbYagThermoCouple.iRaw := TIIB[IM5K2-EL3314-E4]^TC Inputs Channel 2^Value;
                              .fbFlowMeter.iRaw := TIIB[IM5K2-EL3052-E5]^AI Standard Channel 1^Value'}
    fbIM5K2: FB_PPM;
END_VAR


fbIM5K2.stOut.fPosition := -8.92;
fbIM5K2.stOut.bUseRawCounts := FALSE;
fbIM5K2.stOut.bValid := TRUE;
fbIM5K2.stOut.stPMPS.sPmpsState := 'IM5K2:PPM-OUT';

fbIM5K2.stPower.fPosition := -48.02;
fbIM5K2.stPower.bUseRawCounts := FALSE;
fbIM5K2.stPower.bValid := TRUE;
fbIM5K2.stPower.stPMPS.sPmpsState := 'IM5K2:PPM-POWERMETER';

fbIM5K2.stYag1.fPosition := -72.02;
fbIM5K2.stYag1.bUseRawCounts := FALSE;
fbIM5K2.stYag1.bValid := TRUE;
fbIM5K2.stYag1.stPMPS.sPmpsState := 'IM5K2:PPM-YAG1';

fbIM5K2.stYag2.fPosition := -98.03;
fbIM5K2.stYag2.bUseRawCounts := FALSE;
fbIM5K2.stYag2.bValid := TRUE;
fbIM5K2.stYag2.stPMPS.sPmpsState := 'IM5K2:PPM-YAG2';

fbIM5K2(
    fbArbiter := GVL.fbArbiter2,
    fbFFHWO := GVL.fbFastFaultOutput2,
    stYStage := Main.M14,
    sDeviceName := 'IM5K2:PPM',
    sTransitionKey := 'IM5K2:PPM-TRANSITION',
    bEnableMotion := TRUE,
    bEnableBeamParams := TRUE,
    bEnablePositionLimits := TRUE,
    fFlowOffset := 0.0,
);

END_PROGRAM

// ---- POUs/PRG_PF2K2_WFS.TcPOU
PROGRAM PRG_PF2K2_WFS
VAR
    {attribute 'pytmc' := '
        pv: PF2K2:WFS
        io: io
    '}
    {attribute 'TcLinkTo' := '.fbThermoCouple1.bError 		:= TIIB[PF2K2-EL3314-E5]^TC Inputs Channel 1^Status^Error;
                              .fbThermoCouple1.bUnderrange	:= TIIB[PF2K2-EL3314-E5]^TC Inputs Channel 1^Status^Underrange;
                              .fbThermoCouple1.bOverrange 	:= TIIB[PF2K2-EL3314-E5]^TC Inputs Channel 1^Status^Overrange;
                              .fbThermoCouple1.iRaw 		:= TIIB[PF2K2-EL3314-E5]^TC Inputs Channel 1^Value;
                              .fbThermoCouple2.bError 		:= TIIB[PF2K2-EL3314-E5]^TC Inputs Channel 2^Status^Error;
                              .fbThermoCouple2.bUnderrange 	:= TIIB[PF2K2-EL3314-E5]^TC Inputs Channel 2^Status^Underrange;
                              .fbThermoCouple2.bOverrange 	:= TIIB[PF2K2-EL3314-E5]^TC Inputs Channel 2^Status^Overrange;
                              .fbThermoCouple2.iRaw 		:= TIIB[PF2K2-EL3314-E5]^TC Inputs Channel 2^Value'}
    fbPF2K2: FB_WFS;

    //stSiBP: ST_BeamParams := PMPS_GVL.cstFullBeam;
END_VAR

(*
   Avoid damage peak between 3.2 keV and 1.6 keV
*)
//stSiBp.neVRange := F_eVExcludeRange(1600, 3200);
// Drop transmission to 20%
//stSiBP.nTran := 0.2;

fbPF2K2.stOut.fPosition := -15.00;
fbPF2K2.stOut.bUseRawCounts := FALSE;
fbPF2K2.stOut.bValid := TRUE;
fbPF2K2.stOut.stPMPS.sPmpsState := 'PF2K2:WFS-OUT';

fbPF2K2.stTarget1.fPosition := -97.789;
fbPF2K2.stTarget1.bUseRawCounts := FALSE;
fbPF2K2.stTarget1.bValid := TRUE;
fbPF2K2.stTarget1.stPMPS.sPmpsState := 'PF2K2:WFS-TARGET1';

fbPF2K2.stTarget2.fPosition := -83.416;
fbPF2K2.stTarget2.bUseRawCounts := FALSE;
fbPF2K2.stTarget2.bValid := TRUE;
fbPF2K2.stTarget2.stPMPS.sPmpsState := 'PF2K2:WFS-TARGET2';

fbPF2K2.stTarget3.fPosition := -69.043;
fbPF2K2.stTarget3.bUseRawCounts := FALSE;
fbPF2K2.stTarget3.bValid := TRUE;
fbPF2K2.stTarget3.stPMPS.sPmpsState := 'PF2K2:WFS-TARGET3';

fbPF2K2.stTarget4.fPosition := -54.669;
fbPF2K2.stTarget4.bUseRawCounts := FALSE;
fbPF2K2.stTarget4.bValid := TRUE;
fbPF2K2.stTarget4.stPMPS.sPmpsState := 'PF2K2:WFS-TARGET4';

fbPF2K2.stTarget5.fPosition := -40.296;
fbPF2K2.stTarget5.bUseRawCounts := FALSE;
fbPF2K2.stTarget5.bValid := TRUE;
fbPF2K2.stTarget5.stPMPS.sPmpsState := 'PF2K2:WFS-TARGET5';

fbPF2K2(
    fbArbiter := GVL.fbArbiter2,
    fbFFHWO := GVL.fbFastFaultOutput2,
    stYStage := Main.M22,
    stZStage := Main.M23,
    sDeviceName := 'PF2K2:WFS',
    sTransitionKey := 'PF2K2:WFS-TRANSITION',
    bEnableMotion := TRUE,
    bEnableBeamParams := TRUE,
    bEnablePositionLimits := TRUE,
);

END_PROGRAM

// ---- POUs/PRG_TM1K2_ATM.TcPOU
PROGRAM PRG_TM1K2_ATM
VAR
    {attribute 'pytmc' := '
        pv: TM1K2:ATM
        io: io
    '}
    {attribute 'TcLinkTo' := '.fbThermoCouple1.bError := TIIB[TM1K2-EL3314-E5]^TC Inputs Channel 1^Status^Error;
                              .fbThermoCouple1.bUnderrange := TIIB[TM1K2-EL3314-E5]^TC Inputs Channel 1^Status^Underrange;
                              .fbThermoCouple1.bOverrange := TIIB[TM1K2-EL3314-E5]^TC Inputs Channel 1^Status^Overrange;
                              .fbThermoCouple1.iRaw := TIIB[TM1K2-EL3314-E5]^TC Inputs Channel 1^Value'}
    fbTM1K2: FB_ATM;
END_VAR


fbTM1K2.stOut.fPosition := -16;
fbTM1K2.stOut.bUseRawCounts := FALSE;
fbTM1K2.stOut.bValid := TRUE;
fbTM1K2.stOut.stPMPS.sPmpsState := 'TM1K2:ATM-OUT';

fbTM1K2.stTarget1.fPosition := -39.124;
fbTM1K2.stTarget1.bUseRawCounts := FALSE;
fbTM1K2.stTarget1.bValid := TRUE;
fbTM1K2.stTarget1.stPMPS.sPmpsState := 'TM1K2:ATM-TARGET1';

fbTM1K2.stTarget2.fPosition := -53.5;
fbTM1K2.stTarget2.bUseRawCounts := FALSE;
fbTM1K2.stTarget2.bValid := TRUE;
fbTM1K2.stTarget2.stPMPS.sPmpsState := 'TM1K2:ATM-TARGET2';

fbTM1K2.stTarget3.fPosition := -67.874;
fbTM1K2.stTarget3.bUseRawCounts := FALSE;
fbTM1K2.stTarget3.bValid := TRUE;
fbTM1K2.stTarget3.stPMPS.sPmpsState := 'TM1K2:ATM-TARGET3';

fbTM1K2.stTarget4.fPosition := -82.25;
fbTM1K2.stTarget4.bUseRawCounts := FALSE;
fbTM1K2.stTarget4.bValid := TRUE;
fbTM1K2.stTarget4.stPMPS.sPmpsState := 'TM1K2:ATM-TARGET4';

fbTM1K2.stTarget5.fPosition := -96.623;
fbTM1K2.stTarget5.bUseRawCounts := FALSE;
fbTM1K2.stTarget5.bValid := TRUE;
fbTM1K2.stTarget5.stPMPS.sPmpsState := 'TM1K2:ATM-TARGET5';

fbTM1K2(
    fbArbiter := GVL.fbArbiter2,
    fbFFHWO := GVL.fbFastFaultOutput2,
    stYStage := Main.M9,
    stXStage := Main.M10,
    sDeviceName := 'TM1K2:ATM',
    sTransitionKey := 'TM1K2:ATM-TRANSITION',
    bEnableMotion := TRUE,
    bEnableBeamParams := TRUE,
    bEnablePositionLimits := TRUE,
);

END_PROGRAM
